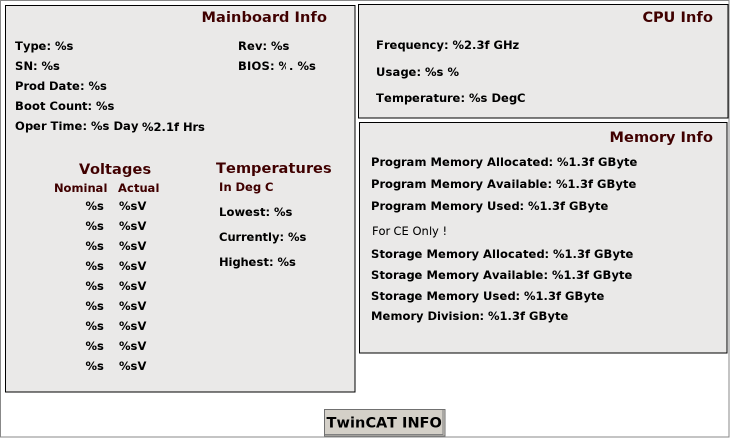
VISUALIZATION MDP_MainboardCPUMemory  // 730x438
    RoundedRectangle (358,4 370x114)
    RoundedRectangle (5,5 350x387)
    Label (192,4 145x26), "Mainboard Info"
    Rectangle (12,35 141x22), "Type: %s", text variable: g_sHMI_MainboardType
    Rectangle (12,55 171x22), "SN: %s", text variable: g_sHMI_MainboardSN
    Rectangle (12,75 207x22), "Prod Date: %s", text variable: g_sHMI_MainboardProdDate
    Rectangle (12,95 151x22), "Boot Count: %s", text variable: g_udiHMI_MainboardBootCount
    Rectangle (12,115 184x22), "Oper Time: %s Days", text variable: g_udiHMI_MainboardOperTimeDays
    Rectangle (139,116 70x22), "%2.1f Hrs", text variable: g_lrHMI_MainboardOperTimeHrs
    Label (213,155 120x26), "Temperatures"
    Rectangle (216,201 102x22), "Lowest: %s", text variable: g_diHMI_MainboardMinTemp
    Rectangle (216,226 102x22), "Currently: %s", text variable: g_iHMI_MainboardActualTemp
    Rectangle (216,251 102x22), "Highest: %s", text variable: g_diHMI_MainboardMaxTemp
    Rectangle (235,35 67x22), "Rev: %s", text variable: g_bHMI_MainboardRevision
    Rectangle (235,55 67x22), "BIOS: %s", text variable: g_bHMI_MainboardBiosMajVers
    Rectangle (286,55 67x22), ". %s", text variable: g_bHMI_MainboardBiosMinVers
    Label (51,175 76x26), "Nominal"
    Rectangle (37,195 70x22), "%s", text variable: g_sHMI_Mainboard1p05v
    Rectangle (37,215 70x22), "%s", text variable: g_sHMI_MainboardVccCore
    Rectangle (37,235 70x22), "%s", text variable: g_sHMI_Mainboard5v
    Rectangle (37,255 70x22), "%s", text variable: g_sHMI_Mainboard12v
    Rectangle (37,275 70x22), "%s", text variable: g_sHMI_MainboardVBatt
    Rectangle (16,295 91x22), "%s", text variable: g_sHMI_MainboardPwrCtrlVcc
    Rectangle (16,315 91x22), "%s", text variable: g_sHMI_MainboardCX2100_5v
    Rectangle (18,335 89x22), "%s", text variable: g_sHMI_MainboardCX2100_12v
    Rectangle (19,355 88x22), "%s", text variable: g_sHMI_MainboardCX2100_24v
    Label (115,175 76x26), "Actual"
    Rectangle (116,195 70x22), "%sV", text variable: g_lrHMI_Mainboard1p05v
    Rectangle (116,215 70x22), "%sV", text variable: g_lrHMI_MainboardVccCore
    Rectangle (116,235 70x22), "%sV", text variable: g_lrHMI_Mainboard5v
    Rectangle (116,255 70x22), "%sV", text variable: g_lrHMI_Mainboard12v
    Rectangle (116,275 70x22), "%sV", text variable: g_lrHMI_MainboardVBatt
    Rectangle (116,295 91x22), "%sV", text variable: g_lrHMI_MainboardPwrCtrlVcc
    Rectangle (116,315 91x22), "%sV", text variable: g_lrHMI_MainboardCX2100_5v
    Rectangle (116,335 89x22), "%sV", text variable: g_lrHMI_MainboardCX2100_12v
    Rectangle (116,355 88x22), "%sV", text variable: g_lrHMI_MainboardCX2100_24v
    Label (76,156 81x26), "Voltages"
    Label (216,174 120x26), "In Deg C"
    Label (596,4 120x26), "CPU Info"
    Rectangle (373,34 163x22), "Frequency: %2.3f GHz", text variable: g_lrHMI_CPUfrequency
    Rectangle (373,61 122x22), "Usage: %s %", text variable: g_iHMI_CPUusage
    Rectangle (373,87 156x22), "Temperature: %s DegC", text variable: g_iHMI_CPUtemperature
    Button (324,409 121x27), "TwinCAT INFO"
        OnMouseClick: change screen: TwinCAT_INFO
    RoundedRectangle (359,122 368x231)
    Label (596,124 120x26), "Memory Info"
    Rectangle (368,151 289x22), "Program Memory Allocated: %1.3f GByte", text variable: g_lrHMI_ProgMemAllocated_InGB
    Rectangle (368,173 287x22), "Program Memory Available: %1.3f GByte", text variable: g_lrHMI_ProgMemAvailable_InGB
    Rectangle (368,243 289x22), "Storage Memory Allocated: %1.3f GByte", text variable: g_lrHMI_ProgStorAllocated_InGB
    Rectangle (368,264 289x22), "Storage Memory Available: %1.3f GByte", text variable: g_lrHMI_ProgStorAvailable_InGB
    Rectangle (368,305 289x22), "Memory Division: %1.3f GByte", text variable: g_lrHMI_ProgStorMemDivision_InGB
    Label (369,216 150x30), "For CE Only !"
    Rectangle (368,195 287x22), "Program Memory Used: %1.3f GByte", text variable: g_lrHMI_ProgMemUsed_InGB
    Rectangle (368,285 289x22), "Storage Memory Used: %1.3f GByte", text variable: g_lrHMI_ProgStorUsed_InGB
END_VISUALIZATION

(* stored: Version 1.1.0.1, ProductVersion 3.1.0.19
   Visu MDP_MainboardCPUMemory: Id {aa1ea548-e7e2-4e83-92ee-4b5205908f91} *)
